FUNCTION_BLOCK FB_LAST_LREAL (* Returns the last value until the R event is triggered. *)
  (* Standard: 61499-2 *)
  (* Version 1.0, 2017-08-28, Marc Jakobi, HTW Berlin *)
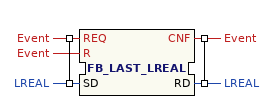
  EVENT_INPUT
    REQ WITH SD; (* Normal Execution Request *)
    R; (* Reset event *)
  END_EVENT
  EVENT_OUTPUT
    CNF WITH RD; (* Execution Confirmation *)
  END_EVENT
  VAR_INPUT
    SD : LREAL; (* Input data *)
  END_VAR
  VAR_OUTPUT
    RD : LREAL; (* Output data *)
  END_VAR
  VAR
    LASTOUTPUT : LREAL; (* Internal Variable *)
    RETURNCURRENTOUTPUT : BOOL := TRUE; (* Internal Variable *)
  END_VAR
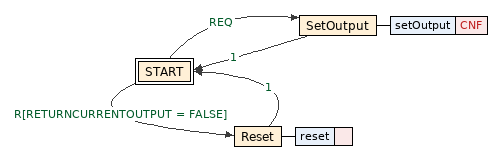
  EC_STATES
    START; (* Initial State *)
    SetOutput : setOutput -> CNF;
    Reset : reset;
  END_STATES
  EC_TRANSITIONS
    START TO SetOutput := REQ;
    SetOutput TO START := 1;
    START TO Reset := R[RETURNCURRENTOUTPUT = FALSE];
    Reset TO START := 1;
  END_TRANSITIONS
  ALGORITHM setOutput IN ST: (* Sets the output *)
IF RETURNCURRENTOUTPUT THEN
	LASTOUTPUT := SD;
	RETURNCURRENTOUTPUT := FALSE;
END_IF;
RD := LASTOUTPUT;
  END_ALGORITHM
  ALGORITHM reset IN ST: (* Resets the FB *)
RETURNCURRENTOUTPUT := TRUE;
  END_ALGORITHM
END_FUNCTION_BLOCK
